FUNCTION ClearDataAnyType : BOOL
VAR_INPUT
	data : __SYSTEM.AnyType;
END_VAR

MEMSET(destAddr := data.pValue, fillByte := 0, n := TO_UDINT(data.diSize));

END_FUNCTION

(* stored: Version 1.1.0.1
   POU ClearDataAnyType: Id {a0da5692-442f-0663-2df4-db9eda984823}, SpecialFunc None *)
